// TIA Portal V16 export
// export: Created 2021-11-12T13:31:57.1506Z, ExportSetting WithDefaults, DisplayName Totally Integrated Automation Portal, DisplayVersion V16 Update 3, DisplayName TIA Portal Version Control Interface, DisplayVersion V16 Update 2, DisplayName TIA Portal Openness, DisplayVersion V16 Update 3, DisplayName SINAMICS Startdrive Advanced, DisplayVersion V16 Update 5, DisplayName SINAMICS Startdrive G130, G150, S120, S150, SINAMICS MV, S210, DisplayVersion V16 Update 5, DisplayName SINAMICS Startdrive G110M, G120, G120C, G120D, G120P, G115D, DisplayVersion V16 Update 5, DisplayName STEP 7 Professional, DisplayVersion V16 Update 3, DisplayName STEP 7 Safety, DisplayVersion V16, DisplayName WinCC UA Professional, DisplayVersion V16 Update 3
DATA_BLOCK "STATUS_000+UC20"   // DB184
{ S7_Optimized_Access := 'TRUE' }
VERSION : 0.1
// stored: AutoNumber true, DBAccessibleFromOPCUA true, IsOnlyStoredInLoadMemory false, IsRetainMemResEnabled false, IsWriteProtectedInAS false, MemoryReserve 100
   VAR
      xxxxx___BinarySensors___xxxxx : Byte;
      xxxxx___BinaryOthers___xxxxx : Byte;
      FB21_14 : Bool;   // 230V Osvětlení rozvaděče se zásuvkou je OK
      FC21_14 : Bool;   // 230V Chlazeni rozvaděče je OK
      EC01_3 : Bool;   // Chlazení rozvaděče je OK
      FC01_14 : Bool;   // 400V Napájení 24V DC je OK
      TB01_14 : Bool;   // Napájení 24V DC je OK
      FC30_14 : Bool;   // 24V Distribuce je OK
      FC30_24 : Bool;   // 24V Distribuce 90 >% zatížení
      FC50_14 : Bool;   // 24V Distribuce je OK
      FC50_24 : Bool;   // 24V Distribuce 90 >% zatížení
      xxxxx___InterfaceSignals___xxxxx : Byte;
      SumErr : Bool;   // Sum of significant errors
      PwrOK : Bool;   // Significant switches ON
      xxxxx___AnalogueSensors___xxxxx : Byte;
      xxxxx___Drives___xxxxx : Byte;
      xxxxx___Other___xxxxx : Byte;
      xxxxx__Alarms___xxxxx : Byte;
      FB21_15 : Struct   // 230V Distributor lightning is OK / 230V Osvětlení rozvaděče se zásuvkou je OK
         Main { S7_SetPoint := 'True'} : "UDT_Status_main";
         Specific { S7_SetPoint := 'True'} : "UDT_DI_Mon_Status_specific";
         Error { S7_SetPoint := 'True'} : "UDT_Error01";
      END_STRUCT;
      FC21_15 : Struct   // 230V Distributor cooling is OK / 230V Chlazeni rozvaděče je OK
         Main { S7_SetPoint := 'True'} : "UDT_Status_main";
         Specific { S7_SetPoint := 'True'} : "UDT_DI_Mon_Status_specific";
         Error { S7_SetPoint := 'True'} : "UDT_Error01";
      END_STRUCT;
      EC01_4 : Struct   // Distributor cooling is OK / Chlazení rozvaděče je OK
         Main { S7_SetPoint := 'True'} : "UDT_Status_main";
         Specific { S7_SetPoint := 'True'} : "UDT_DI_Mon_Status_specific";
         Error { S7_SetPoint := 'True'} : "UDT_Error01";
      END_STRUCT;
      FC01_15 : Struct   // 400V Power supply 24V DC is OK / 400V Napájení 24V DC je OK
         Main { S7_SetPoint := 'True'} : "UDT_Status_main";
         Specific { S7_SetPoint := 'True'} : "UDT_DI_Mon_Status_specific";
         Error { S7_SetPoint := 'True'} : "UDT_Error01";
      END_STRUCT;
      TB01_15 : Struct   // Power supply 24V DC is OK / Napájení 24V DC je OK
         Main { S7_SetPoint := 'True'} : "UDT_Status_main";
         Specific { S7_SetPoint := 'True'} : "UDT_DI_Mon_Status_specific";
         Error { S7_SetPoint := 'True'} : "UDT_Error01";
      END_STRUCT;
      FC30_15 : Struct   // 24V Distribution is OK / 24V Distribuce je OK
         Main { S7_SetPoint := 'True'} : "UDT_Status_main";
         Specific { S7_SetPoint := 'True'} : "UDT_DI_Mon_Status_specific";
         Error { S7_SetPoint := 'True'} : "UDT_Error01";
      END_STRUCT;
      FC30_25 : Struct   // 24V Distribution 90 >% load / 24V Distribuce 90 >% zatížení
         Main { S7_SetPoint := 'True'} : "UDT_Status_main";
         Specific { S7_SetPoint := 'True'} : "UDT_DI_Mon_Status_specific";
         Error { S7_SetPoint := 'True'} : "UDT_Error01";
      END_STRUCT;
      FC50_15 : Struct   // 24V Distribution is OK / 24V Distribuce je OK
         Main { S7_SetPoint := 'True'} : "UDT_Status_main";
         Specific { S7_SetPoint := 'True'} : "UDT_DI_Mon_Status_specific";
         Error { S7_SetPoint := 'True'} : "UDT_Error01";
      END_STRUCT;
      FC50_25 : Struct   // 24V Distribution 90 >% load / 24V Distribuce 90 >% zatížení
         Main { S7_SetPoint := 'True'} : "UDT_Status_main";
         Specific { S7_SetPoint := 'True'} : "UDT_DI_Mon_Status_specific";
         Error { S7_SetPoint := 'True'} : "UDT_Error01";
      END_STRUCT;
   END_VAR
BEGIN
END_DATA_BLOCK
